TEXTLIST TL_RecipesManagerStatus
  0 = 'Idle'
  10 = 'Initialization'
  20 = 'Create'
  30 = 'Load'
  40 = 'Read'
  50 = 'Reload'
  60 = 'Backup'
  70 = 'Restore'
  -10 = 'Abort'
   = ''
END_TEXTLIST

(* stored: Version 1.1.0.1, ProductVersion 3.1.4024.12
   TextList TL_RecipesManagerStatus: Id {1c4e3353-5e75-4c97-97e2-9d418f5b12ce} *)
